// TIA Portal V20 export
DATA_BLOCK "DB_OPC_Axis"   // DB102
{ S7_Optimized_Access := 'TRUE' }
// stored: MemoryReserve 100
   VAR
      ActualValues : Struct
         NumberOfAxes { S7_SetPoint := 'True'} : DInt;
         Axes : Array[0..100] of "UDT_OPC_ActualValuesAxis";
      END_STRUCT;
      TaughtPositions : Struct
         NumberOfItems { S7_SetPoint := 'True'} : DInt;
         Items : Array[0..100] of "UDT_OPC_TaughtPositionsItems";
      END_STRUCT;
      Teach : Struct
         Buttons : Struct
            Teach : "UDT_OPCButtons";
         END_STRUCT;
         Parameters : Struct
            AxisId : DInt;
            PositionId : DInt;
         END_STRUCT;
         Current : Struct
            ActualPosition : LReal;
            TaughtPosition : LReal;
         END_STRUCT;
      END_STRUCT;
   END_VAR
BEGIN
END_DATA_BLOCK
